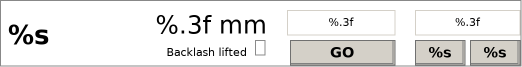
VISUALIZATION VISU_M2AxisControl  // 522x67
VAR_IN_OUT
	widget : M2AxisWidget;
END_VAR
    Rectangle (5,10 90x50), "%s", text variable: widget.name
    Rectangle (105,10 165x30), "%.3f mm", text variable: widget.position_mm
        p55702900: widget.poweredTextColor
    Textfield (287,10 108x25), "%.3f", text variable: widget.absolute_setpoint
        OnMouseClick: write the text variable via VisuDialogs.Numpad, title 'Enter the absolute position setpoint in mm'
    Textfield (415,10 105x25), "%.3f", text variable: widget.relative_setpoint
        OnMouseClick: write the text variable via VisuDialogs.Numpad, title 'Enter the relative position offset in mm'
    Button (290,40 105x25), "GO", input disabled if: widget.absolute_go_disabled
        OnMouseClick: execute { widget.absolute_go := TRUE; }
    Button (415,40 50x25), "%s", text variable: widget.relative_goLeft_text, input disabled if: widget.relative_goLeft_disabled
        OnMouseClick: execute { widget.relative_goLeft := TRUE; }
    Button (470,40 50x25), "%s", text variable: widget.relative_goRight_text, input disabled if: widget.relative_goRight_disabled
        OnMouseClick: execute { widget.relative_goRight := TRUE; }
    Frame (255,40 10x15)
        shows VISU_State_gray_green(state := widget.backlashLifted)
    Label (100,40 150x25), "Backlash lifted"
END_VISUALIZATION

(* stored: Version 1.1.0.1, ProductVersion 3.1.4019.2
   Visu VISU_M2AxisControl: Id {0d52d8be-19e4-47a1-aad0-ea77036eb418} *)
